(*

.. <legal notes>

legal notes
=================
| SPDX-FileCopyrightText: © 2025 Oleksandr Tiutyk <trofimich@gmail.com>
| SPDX-License-Identifier: LGPL-3.0-only
| For details check: LGPL-3.0-only_

.. _LGPL-3.0-only: https://www.gnu.org/licenses/lgpl-3.0.en.html

.. </legal notes>

*)

{attribute 'no_explicit_call' := 'do not call this function block directly'} 
{attribute 'enable_dynamic_creation'}
FUNCTION_BLOCK SequenceActivity EXTENDS Activity IMPLEMENTS ISequenceActivity
VAR
	{attribute 'OPC.UA.DA' := '0'}
	_ClassName : STRING := __POUNAME();

	{attribute 'OPC.UA.DA' := '0'}
	_Children : Collections.List(0);

	{attribute 'OPC.UA.DA' := '0'}
	_CurrentActivityIndex : DINT := -1;
END_VAR

METHOD AddChildActivity
VAR_INPUT
	activity : IActivity;
END_VAR
VAR
	argumentNullExcxeption : Core.ArgumentNullException;
END_VAR
IF activity = 0  THEN
	argumentNullExcxeption.Throw(NamespaceName, ClassName, __POUNAME(), __POSITION(), 'activity');
END_IF

activity.Parent := THIS^;

_Children.AppendGeneric(Core.GenericValueFactory.FromParts(GENERIC_TYPE_CLASS.TYPE_OBJECT, activity.Address, activity.Size, GENERIC_MEMORY_MANAGEMENT_BEHAVIOR.STORE_ORIGINAL_REFERENCE_AND_NOT_OWNS_MEMORY));
END_METHOD

{attribute 'monitoring' := 'call'}
PROPERTY ClassName : STRING
GET
ClassName := _ClassName;
END_GET
END_PROPERTY

{attribute 'monitoring' := 'call'}
PROPERTY FINAL CurrentActivity : IActivity
GET
IF _Children.Count > 0 AND_THEN _CurrentActivityIndex >= 0 AND_THEN _CurrentActivityIndex < _Children.Count THEN
	__QUERYINTERFACE(_Children.Get(_CurrentActivityIndex).AsObject(), CurrentActivity);
END_IF
END_GET
END_PROPERTY

{attribute 'monitoring' := 'call'}
PROPERTY FINAL CurrentActivityIndex : DINT
GET
CurrentActivityIndex := _CurrentActivityIndex;
END_GET
END_PROPERTY

{attribute 'monitoring' := 'call'}
PROPERTY NamespaceName : STRING
GET
NamespaceName := CurrentNamespace.Name;
END_GET
END_PROPERTY

METHOD PROTECTED OnAborting 
VAR_INPUT
	isStart : BOOL;
END_VAR
VAR_OUTPUT
	done : BOOL;
END_VAR
VAR
	activity : IActivity;
END_VAR
IF _Children.Count < 1 THEN
	done := TRUE;
	RETURN;
END_IF

activity := CurrentActivity;

IF activity = 0 OR_ELSE NOT activity.Busy THEN
	done := TRUE;
	RETURN;
END_IF

IF isStart THEN
	activity.StartAbort();
ELSE
	activity.Execute();
END_IF

done := NOT activity.Busy;
END_METHOD

METHOD PROTECTED OnRunning 
VAR_INPUT
	isStart : BOOL;
END_VAR
VAR_OUTPUT
	done : BOOL;
END_VAR
VAR
	activity : IActivity;
	
	currentActivityIsNullException : Core.NullReferenceException;
END_VAR
IF _Children.Count < 1 THEN
	done := TRUE;
	RETURN;
END_IF

IF isStart AND_THEN _CurrentActivityIndex < 0 THEN
	_CurrentActivityIndex := 0;
END_IF

activity := CurrentActivity;

IF activity = 0 THEN
	currentActivityIsNullException.Throw(NamespaceName, ClassName, __POUNAME(), __POSITION(), 'CurrentActivity');
END_IF

IF isStart OR_ELSE NOT activity.Busy THEN
	activity.Start();
ELSE
	activity.Execute();
END_IF

IF NOT activity.Busy THEN
	selectNextTask();
END_IF

done := _CurrentActivityIndex < 0;
END_METHOD

METHOD PRIVATE selectNextTask
IF _CurrentActivityIndex < _Children.Count - 1 THEN
	_CurrentActivityIndex := _CurrentActivityIndex + 1;
ELSE	
	_CurrentActivityIndex := -1;
END_IF
END_METHOD

{attribute 'monitoring' := 'call'}
PROPERTY Size : ULINT
GET
Size := XSIZEOF(THIS^);
END_GET
END_PROPERTY

END_FUNCTION_BLOCK

(* stored: Version 1.1.0.1
   POU SequenceActivity: Id {5f2d9604-eb7b-45e3-84bc-b901136bbe0b}, SpecialFunc None
   Folder Overriden: Id {1b1c5863-9f32-4a15-87e0-d0e2df5c3f78}
   Folder Service members: Id {1f0247af-e697-46d2-a7ad-83444186c8c6}
   Method AddChildActivity: Id {2c396587-941c-45cd-a7de-a236bec55a27}
   Property ClassName: Id {ba95610f-5219-47c9-8c57-311d9e60e72f}
   Get Get: Id {013b3af7-a06d-4fbf-a280-1144598a7235}
   Property CurrentActivity: Id {c0d02002-6e75-4b84-a496-ad82ebf3d647}
   Get Get: Id {28df5953-696c-4fdc-b8d7-69723340165e}
   Property CurrentActivityIndex: Id {57ee575b-1867-4622-b68b-c137e6c21192}
   Get Get: Id {c24f3d90-442c-4a36-a32c-a9f9b1ca1fa1}
   Property NamespaceName: Id {770d34c9-dbf7-4149-9b56-f9dd9d652c8b}
   Get Get: Id {7d1a0f6f-5dcd-4e0e-aac5-a3ff24ac9579}
   Method OnAborting: Id {3a5ab894-6d0b-4ec0-b72f-2b4254f65f95}
   Method OnRunning: Id {2c7c0cfd-db41-4ccf-92fc-38a7fc6a065c}
   Method selectNextTask: Id {158fb674-f3c7-4b23-a12c-a74041bb8e97}
   Property Size: Id {b289e881-1f3e-4abc-9a70-4494d509b71b}
   Get Get: Id {40179bbc-4746-4890-bbcf-233fb2a96bdf} *)
